INTERFACE I_ExceptionHandling

METHOD BuildException : ST_Exception
VAR_INPUT
	eException : E_Exception;
END_VAR
END_METHOD

METHOD Catch : BOOL
VAR_INPUT
	eException : E_Exception;
	eExceptionOrigin : E_Origin;
END_VAR
END_METHOD

METHOD ExceptionAvailable : BOOL
VAR_INPUT
END_VAR
END_METHOD

METHOD ForwardToNextLevel : BOOL
VAR_INPUT
	sender : I_ExceptionHandling;
END_VAR
END_METHOD

METHOD GenericCatch : BOOL
VAR_INPUT
	eException : E_Exception;
END_VAR
END_METHOD

PROPERTY getException : ST_Exception
GET
END_GET
END_PROPERTY

PROPERTY getExceptionOrigin : E_Origin
GET
END_GET
END_PROPERTY

METHOD Throw : BOOL
VAR_INPUT
	stException : ST_Exception;
END_VAR
END_METHOD

END_INTERFACE

(* stored: Version 1.1.0.1, ProductVersion 3.1.4024.0
   Itf I_ExceptionHandling: Id {d05c4919-1dbf-49ef-81be-1eb3c31fdd6c}
   Method BuildException: Id {1b1d43bd-261c-4d6b-bccf-fae29ab4e826}
   Method Catch: Id {547f77b8-3bae-446f-a966-eaa2371e4ff2}
   Method ExceptionAvailable: Id {5ebfad5f-abc0-4515-aeb4-06e73d73a23b}
   Method ForwardToNextLevel: Id {7b5e33b6-5025-4e95-9822-b466a812f28e}
   Method GenericCatch: Id {6546e87b-6ce2-4c7e-b984-19a451fd56f3}
   Property getException: Id {7185c56b-9383-443e-9d5b-6f3e5687528c}
   Get Get: Id {417c9224-cbcb-4676-84b6-0cc373878cc9}
   Property getExceptionOrigin: Id {ea4e7814-b1ed-457d-8fb2-a18aa4a80c13}
   Get Get: Id {49294241-bf64-4e7a-8649-e823e91b4e7f}
   Method Throw: Id {b48f5560-29b3-4065-8aa9-a96e5d54929b} *)
